FUNCTION_BLOCK FB_HbotHome
VAR_INPUT
	bExecute : BOOL;
	Velocity : REAL;
END_VAR
VAR_OUTPUT
	bDone : BOOL;
	bError : BOOL;
	bBusy : BOOL;
END_VAR
VAR
	init : R_TRIG;
	StepperAJog : MC_Jog;
	StepperBJog : MC_Jog;
	
	StepperASetPos : MC_SetPosition;
	StepperBSetPos : MC_SetPosition;
	
	StepperAHome : MC_Home;
	StepperBHome : MC_Home;
	
	StepperAHalt : MC_Halt;
	StepperBHalt : MC_Halt;
	
	homeSequence : (homeX, homeY, halt, forcecalibration, done, error);
	ErrorTimeout : ton;
	ErrorTimeoutCase : INT;
END_VAR
VAR_IN_OUT
	StepperA	:	AXIS_REF;
	StepperB	:	AXIS_REF;
	
	limitSwitchX : BOOL;
	limitSwitchY : BOOL;
END_VAR

init(CLK := bExecute); // detect rising edge

IF bExecute AND NOT bError THEN 
	IF init.Q THEN // if it is on rising edge (i.e, first instance of bexecute is true
		homeSequence := homeX; // set switch case to homeX
	END_IF
	
	CASE homeSequence OF
	homeX :
		bBusy := TRUE;
		bDone := FALSE;
		// Home Cartesian X, Both steppers to jog forward at the same speed
		StepperAJog(Axis := StepperA, JogForward := TRUE, Velocity := Velocity);
		StepperBJog(Axis := StepperB, JogForward := TRUE, Velocity := Velocity);
		IF StepperAJog.Error OR StepperBJog.Error THEN
			homeSequence := error;
		END_IF
		IF limitSwitchX THEN // if limit switch is triggered, stop jogging and go to homeY case
			StepperAJog(Axis := StepperA, JogForward := FALSE);
			StepperBJog(Axis := StepperB, JogForward := FALSE);
			homeSequence := homeY;
		END_IF
		IF StepperAJog.CommandAborted OR StepperBJog.CommandAborted THEN 
			homeSequence := Error;
		END_IF
	
	homeY :
		// Home Cartesian Y, Both steppers to jog in opposite directions at the same speed
		StepperAJog(Axis := StepperA, JogForward := TRUE, Velocity := Velocity);
		StepperBJog(Axis := StepperB, JogBackwards := TRUE, Velocity := Velocity);
		IF StepperAJog.Error OR StepperBJog.Error THEN
			homeSequence := error;
		END_IF
		IF limitSwitchY THEN // if limit switch is triggered, stop jogging and go to halt case
			StepperAJog(Axis := StepperA, JogForward := FALSE);
			StepperBJog(Axis := StepperB, JogBackwards := FALSE);
			homeSequence := halt;
		END_IF
		
		IF StepperAJog.CommandAborted OR StepperBJog.CommandAborted THEN 
			homeSequence := Error;
		END_IF
		
	halt :
		// halting motors
		StepperAHalt(Axis := StepperA, Execute := TRUE);
		StepperBHalt(Axis := StepperB, Execute := TRUE);
		IF StepperAHalt.Done AND StepperBHalt.Done THEN
			homeSequence := forcecalibration; // once stopped, reset mc_halt and go to force calibration case
			StepperAHalt(Axis := StepperA, Execute := FALSE);
			StepperBHalt(Axis := StepperB, Execute := FALSE);
		ELSIF StepperAHalt.Error OR StepperBHalt.Error THEN
			homeSequence := error;
		END_IF
		
		
	forcecalibration :
		// set stepper positions to 0
		StepperASetPos(Axis := StepperA, Position := 0.0, Mode := FALSE, Execute := TRUE);
		StepperBSetPos(Axis := StepperB, Position := 0.0, Mode := FALSE, Execute := TRUE);
		IF StepperASetPos.Error OR StepperBSetPos.Error THEN
			homeSequence := error;
		ELSIF StepperASetPos.Done AND StepperBSetPos.Done THEN
			homeSequence := done; // go to done case
			StepperASetPos(Axis := StepperA, Position := 0.0, Mode := FALSE, Execute := FALSE);
			StepperBSetPos(Axis := StepperB, Position := 0.0, Mode := FALSE, Execute := FALSE);
		END_IF
		
	done :
		bDone := TRUE;
		bBusy := FALSE;
		
	error:
	
		CASE ErrorTimeoutCase OF 
		0: bError := TRUE;
		ErrorTimeout (IN := TRUE, PT := T#5000MS);
		IF ErrorTimeout.Q THEN 
			ErrorTimeoutCase := 10; 
		END_IF
		10: bError := FALSE; 
		homeSequence := done;
		ErrorTimeoutCase := 0; 
		
		END_CASE
		
	END_CASE
ELSE
	bDone := FALSE;
END_IF

END_FUNCTION_BLOCK

(* stored: Version 1.1.0.1, ProductVersion 3.1.4024.12
   POU FB_HbotHome: Id {211248de-5d88-41dd-be9c-3250d67eb550}, SpecialFunc None *)
